SUBAPPLICATION Uebung_091 (* Beispiel für E_TRAIN *)
  (* Standard: 61499-2; Description: Copyright (c) 2023 Meisterschulen am Ostbahnhof This program and the accompanying materials are made available under the terms of the Eclipse Public License 2.0 which is available at https://www.eclipse.org/legal/epl-2.0/ SPDX-License-Identifier: EPL-2.0 *)
  (* Version 1.0, 2023-10-23, Franz Höpfinger, Meisterschulen am Ostbahnhof *)
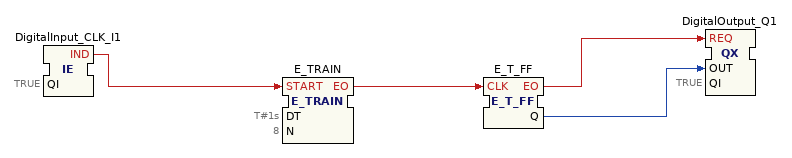
  (* E_TRAIN wird 8 Events ausgeben, das erste 1s nach dem Click, das letzte 8s nach dem Click *)
  FBS
    DigitalOutput_Q1 : QX(QI := TRUE);
    E_TRAIN : E_TRAIN(DT := T#1s, N := 8);
    DigitalInput_CLK_I1 : IE(QI := TRUE);
    E_T_FF : E_T_FF;
  END_FBS
  EVENT_CONNECTIONS
    DigitalInput_CLK_I1.IND TO E_TRAIN.START;
    E_TRAIN.EO TO E_T_FF.CLK;
    E_T_FF.EO TO DigitalOutput_Q1.REQ;
  END_CONNECTIONS
  DATA_CONNECTIONS
    E_T_FF.Q TO DigitalOutput_Q1.OUT;
  END_CONNECTIONS
END_SUBAPPLICATION
